// TIA Portal V17 export
// export: Created 2024-09-02T12:49:58.0233931Z, ExportSetting WithDefaults, DisplayName Totally Integrated Automation Portal, DisplayVersion V17, DisplayName TIA Portal Openness, DisplayVersion V17, DisplayName TIA Portal Version Control Interface, DisplayVersion V17, DisplayName STEP 7 Professional, DisplayVersion V17, DisplayName STEP 7 Safety, DisplayVersion V17, DisplayName WinCC Professional, DisplayVersion V17
FUNCTION "HLP_HMI_Funktion" : Void   // FC30201, LAD
TITLE = HLP Button / HLP Button
{ S7_Optimized_Access := 'TRUE' }
AUTHOR : OlegFuehrus
FAMILY : HLP
NAME : HLP
VERSION : 1.0
// stored: AutoNumber false, IsIECCheckEnabled false, SetENOAutomatically false, UDAEnableTagReadback false
   VAR_INPUT
      i_FKT : Int;   // Funktionskodierung / Function coding
      i_ON : Bool;   // Funktionsanzeige / function display
      i_ENBL : Bool;   // Funktionsfreigabe / Functional Approve
      i_RMG : Bool;   // Rückmeldung / Feedback
      i_ANF : Bool;   // Anforderung / Requirement
      i_SFK : Bool;   // Sonderfunktion / Special functions
   END_VAR
   VAR_IN_OUT
      io_Button : Struct   // Funktion / Function
         Design : Int;   // Button Anzeige Gestaltung / Button Display Design
         active : Bool;   // Button aktiv (gedrückt) / Button active (pressed)
      END_STRUCT;
   END_VAR
   VAR_TEMP   // added for the SCL form of the ladder/FBD networks
      _w1 : Bool;
   END_VAR
BEGIN

REGION Network 1: Reset button active (pressed) / Button aktiv (gedrückt) zuruecksetzen
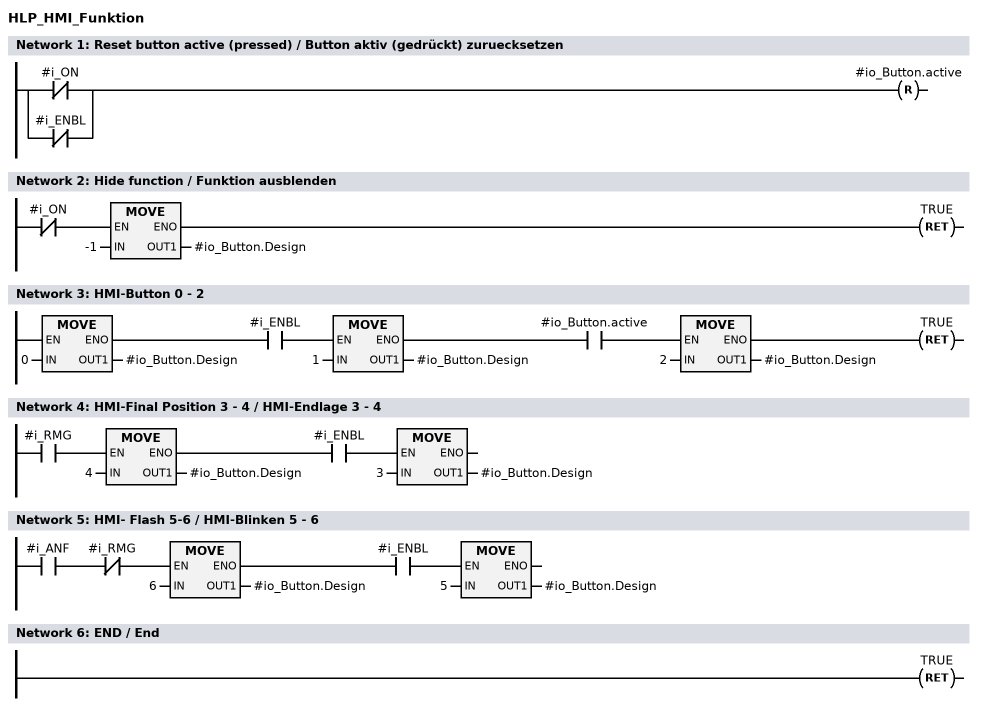
   RUNG wire#powerrail
      I_Contact( #i_ON )
      wire#w1
      R_Coil( #io_Button.active )
   END_RUNG
   RUNG wire#powerrail
      I_Contact( #i_ENBL )
   END_RUNG wire#w1
   // the same network as SCL:
   IF NOT #i_ON OR NOT #i_ENBL THEN #io_Button.active := FALSE; END_IF;
END_REGION

REGION Network 2: Hide function / Funktion ausblenden
   RUNG wire#powerrail
      I_Contact( #i_ON )
      Move(in := -1, out1 => #io_Button.Design)
      ReturnCoil( TRUE )
   END_RUNG
   // the same network as SCL:
   IF NOT #i_ON THEN
       #io_Button.Design := -1;
       ENO := TRUE;
       RETURN;
   END_IF;
END_REGION

REGION Network 3: HMI-Button 0 - 2
   RUNG wire#powerrail
      Move(in := 0, out1 => #io_Button.Design)
      Contact( #i_ENBL )
      Move(in := 1, out1 => #io_Button.Design)
      Contact( #io_Button.active )
      Move(in := 2, out1 => #io_Button.Design)
      ReturnCoil( TRUE )
   END_RUNG
   // the same network as SCL:
   #io_Button.Design := 0;
   IF #i_ENBL THEN #io_Button.Design := 1; END_IF;
   #_w1 := #i_ENBL AND #io_Button.active;
   IF #_w1 THEN
       #io_Button.Design := 2;
       ENO := TRUE;
       RETURN;
   END_IF;
END_REGION

REGION Network 4: HMI-Final Position 3 - 4 / HMI-Endlage 3 - 4
   RUNG wire#powerrail
      Contact( #i_RMG )
      Move(in := 4, out1 => #io_Button.Design)
      Contact( #i_ENBL )
      Move(in := 3, out1 => #io_Button.Design)
   END_RUNG
   // the same network as SCL:
   IF #i_RMG THEN #io_Button.Design := 4; END_IF;
   IF #i_RMG AND #i_ENBL THEN #io_Button.Design := 3; END_IF;
END_REGION

REGION Network 5: HMI- Flash 5-6 / HMI-Blinken 5 - 6
   RUNG wire#powerrail
      Contact( #i_ANF )
      I_Contact( #i_RMG )
      Move(in := 6, out1 => #io_Button.Design)
      Contact( #i_ENBL )
      Move(in := 5, out1 => #io_Button.Design)
   END_RUNG
   // the same network as SCL:
   #_w1 := #i_ANF AND NOT #i_RMG;
   IF #_w1 THEN #io_Button.Design := 6; END_IF;
   IF #_w1 AND #i_ENBL THEN #io_Button.Design := 5; END_IF;
END_REGION

REGION Network 6: END / End
   RUNG wire#powerrail
      ReturnCoil( TRUE )
   END_RUNG
   // the same network as SCL:
   ENO := TRUE;
   RETURN;
END_REGION
END_FUNCTION
